FUNCTION_BLOCK FB_EventHandler IMPLEMENTS I_EventHandler
VAR_INPUT
END_VAR
VAR_OUTPUT
END_VAR
VAR
	// private instance var's
	iLog			: I_Logger;
	afbAlarm      	: ARRAY[0..Const.iMaxIdxAlam] OF FB_TcAlarm;
	fbCodeErrRef,
	fbAlarmRef      : REFERENCE TO FB_TcAlarm;
	fbMsg			: FB_TcMessage;
	fbEventLogger	: FB_TcEventLogger;
	ISb 			: I_StringBuilder;
	fbInternalSb	: FB_StringBuilder;
	iCntAlm			: INT;
	bInfoActive,
	bWarningActive,
	bErrorActive	: BOOL;
END_VAR

//ToDo: SetJsonAttribute (e.g.: error reaction)
//ToDo: F_GetEventText o.ä.
//ToDo: Listener?

// unit tests
Test();

METHOD PUBLIC ArgAddDint : I_EventHandler
VAR_INPUT
	value : DINT;
END_VAR
ArgAddDint := THIS^;
IF __ISVALIDREF(fbAlarmRef) THEN
	fbAlarmRef.ipArguments.AddDInt(value);
END_IF
END_METHOD

METHOD PUBLIC ArgAddEventRef : I_EventHandler
VAR_INPUT
	value : TcEventEntry;
END_VAR
ArgAddEventRef := THIS^;
IF __ISVALIDREF(fbAlarmRef) THEN
	fbAlarmRef.ipArguments.AddEventReferenceEx(value);
END_IF
END_METHOD

METHOD PUBLIC ArgAddLreal : I_EventHandler
VAR_INPUT
	value : LREAL;
END_VAR
ArgAddLreal := THIS^;
IF __ISVALIDREF(fbAlarmRef) THEN
	fbAlarmRef.ipArguments.AddLReal(value);
END_IF
END_METHOD

METHOD PUBLIC ArgAddString : I_EventHandler
VAR_IN_OUT CONSTANT
	value : STRING;
END_VAR
ArgAddString := THIS^;
IF __ISVALIDREF(fbAlarmRef) THEN
	fbAlarmRef.ipArguments.AddString(value);
END_IF
END_METHOD

METHOD PUBLIC ArgAddWString : I_EventHandler
VAR_IN_OUT CONSTANT
	value : WSTRING;
END_VAR
ArgAddWString := THIS^;
IF __ISVALIDREF(fbAlarmRef) THEN
	fbAlarmRef.ipArguments.AddWString(value);
END_IF
END_METHOD

METHOD PUBLIC ArgClear : I_EventHandler
ArgClear := THIS^;
IF __ISVALIDREF(fbAlarmRef) THEN
	fbAlarmRef.ipArguments.Clear();
END_IF
END_METHOD

METHOD PUBLIC ArgSbAppend : I_EventHandler
VAR_IN_OUT CONSTANT
	value : T_MaxString;
END_VAR
ArgSbAppend := THIS^;

IF ISb <> 0 THEN
	ISb.Append(value);
END_IF
END_METHOD

METHOD PUBLIC ArgSbAppendAny : I_EventHandler
VAR_INPUT
	value : ANY;
END_VAR
ArgSbAppendAny := THIS^;

IF ISb <> 0 THEN
	ISb.AppendAny(value);
END_IF
END_METHOD

METHOD PUBLIC ArgSbAppendAnyRaise : HRESULT
VAR_INPUT
	value : ANY;
END_VAR
ArgSbAppendAnyRaise := ArgSbAppendAny(value).ArgSetSbRaise();
END_METHOD

METHOD PUBLIC ArgSbAppendRaise : HRESULT
VAR_IN_OUT CONSTANT
	value : T_MaxString;
END_VAR
ArgSbAppendRaise := ArgSbAppendSet(value).Raise();
END_METHOD

METHOD PUBLIC ArgSbAppendS : I_EventHandler
VAR_INPUT
	value : T_MaxString := '';
END_VAR
ArgSbAppendS := ArgSbAppend(value);
END_METHOD

METHOD PUBLIC ArgSbAppendSet : I_EventHandler
VAR_IN_OUT CONSTANT
	value : T_MaxString;
END_VAR
ArgSbAppendSet := ArgSbAppend(value).ArgSetSb();
END_METHOD

METHOD PUBLIC ArgSbAppendWs : I_EventHandler
VAR_IN_OUT CONSTANT
	value : WSTRING;
END_VAR
ArgSbAppendWs := THIS^;

IF ISb <> 0 THEN
	ISb.AppendWs(value);
END_IF
END_METHOD

METHOD PUBLIC ArgSbAppendWsRaise : HRESULT
VAR_IN_OUT CONSTANT
	value : WSTRING;
END_VAR
ArgSbAppendWsRaise := ArgSbAppendWs(value).ArgSetSbRaise();
END_METHOD

METHOD PUBLIC ArgSbInit : I_EventHandler
VAR_IN_OUT CONSTANT
	value : T_MaxString;
END_VAR
Isb := fbInternalSb.Set(value);
ArgSbInit := THIS^;
END_METHOD

METHOD PUBLIC ArgSbInitExternal : I_EventHandler
VAR_INPUT
	sb	: I_StringBuilder;
END_VAR
ISb := sb;
ArgSbInitExternal := THIS^;
END_METHOD

METHOD PUBLIC ArgSbInitWs : I_EventHandler
VAR_IN_OUT CONSTANT
	value : WSTRING;
END_VAR
Isb := fbInternalSb.SetWs(value);
ArgSbInitWs := THIS^;
END_METHOD

METHOD PUBLIC ArgSetDint : I_EventHandler
VAR_INPUT
	value : DINT;
END_VAR
ArgSetDint := ArgClear().ArgAddDint(value);
END_METHOD

METHOD PUBLIC ArgSetEventRef : I_EventHandler
VAR_INPUT
	value : TcEventEntry;
END_VAR
ArgSetEventRef := ArgClear().ArgAddEventRef(value);
END_METHOD

METHOD PUBLIC ArgSetLreal : I_EventHandler
VAR_INPUT
	value : LREAL;
END_VAR
ArgSetLreal := ArgClear().ArgAddLreal(value);
END_METHOD

METHOD PUBLIC ArgSetSb : I_EventHandler
VAR_INPUT
	sb 		: I_StringBuilder := 0; // optional external string builder, set to 0 to use internal
END_VAR
VAR
	value	: STRING;
END_VAR
IF sb = 0 THEN
	sb := Isb;
END_IF

value := sb.ToString();
ArgSetSb := ArgClear().ArgAddString(value);
END_METHOD

METHOD PUBLIC ArgSetSbRaise : HRESULT
VAR_INPUT
	sb	: I_StringBuilder := 0; // optional external string builder, set to 0 to use internal
END_VAR
ArgSetSbRaise := ArgSetSb(sb).Raise();
END_METHOD

METHOD PUBLIC ArgSetString : I_EventHandler
VAR_IN_OUT CONSTANT
	value : STRING;
END_VAR
ArgSetString := ArgClear().ArgAddString(value);
END_METHOD

METHOD PUBLIC ArgSetWString : I_EventHandler
VAR_IN_OUT CONSTANT
	value : WSTRING;
END_VAR
ArgSetWString := ArgClear().ArgAddWString(value);
END_METHOD

METHOD PUBLIC CreateAlarm : I_EventHandler
VAR_INPUT
	stEventEntry      : TcEventEntry;
    bWithConfirmation : BOOL := FALSE;
    ipSourceInfo      : I_TcSourceInfo := NULL;
END_VAR
VAR
	hres 	: HRESULT;
	msg		: STRING;
END_VAR
CreateAlarm := THIS^;
IF (iCntAlm > Const.iMaxIdxAlam) THEN
	msg := CONCAT('Max. events exceeded, Const.iMaxIdxAlam: ', TO_STRING(Const.iMaxIdxAlam));
	fbCodeErrRef.ipArguments.Clear().AddString(msg);
	fbCodeErrRef.Raise(0);
	RETURN;
END_IF

hres := afbAlarm[iCntAlm].CreateEx(stEventEntry, bWithConfirmation, ipSourceInfo);

IF (hres = S_OK) THEN
	iCntAlm := iCntAlm + 1;
ELSE
	msg := CONCAT('Create alarm failed, HRESULT: ', TO_STRING(hres));
	fbCodeErrRef.ipArguments.Clear().AddString(msg);
	fbCodeErrRef.Raise(0);
END_IF
END_METHOD

{attribute 'monitoring' := 'call'}
PROPERTY ErrorActive : BOOL
GET
ErrorActive := bErrorActive;
END_GET
END_PROPERTY

{attribute 'monitoring' := 'call'}
PROPERTY InfoActive : BOOL
GET
InfoActive := bInfoActive;
END_GET
END_PROPERTY

METHOD Init : BOOL
iLog := SERVICES.ILog;

// init alarm event classes
CreateAlarm(TC_Events.InternalEventClass.InfoEvent);
CreateAlarm(TC_Events.InternalEventClass.WarningEvent, TRUE);
CreateAlarm(TC_Events.InternalEventClass.ErrorEvent, TRUE);
CreateAlarm(TC_Events.CodeEventClass.InfoEvent);
CreateAlarm(TC_Events.CodeEventClass.WarningEvent, TRUE);
CreateAlarm(TC_Events.CodeEventClass.ErrorEvent, TRUE);
CreateAlarm(TC_Events.SystemEventClass.InfoEvent);
CreateAlarm(TC_Events.SystemEventClass.WarningEvent, TRUE);
CreateAlarm(TC_Events.SystemEventClass.ErrorEvent, TRUE);
CreateAlarm(TC_Events.EtherCatEventClass.InfoEvent);
CreateAlarm(TC_Events.EtherCatEventClass.WarningEvent, TRUE);
CreateAlarm(TC_Events.EtherCatEventClass.ErrorEvent, TRUE);
CreateAlarm(TC_Events.EtherCatEventClass.DevicStateErrorEvent, TRUE);
CreateAlarm(TC_Events.EtherCatEventClass.LinkStateErrorEvent, TRUE);
CreateAlarm(TC_Events.HardwareEventClass.InfoEvent);
CreateAlarm(TC_Events.HardwareEventClass.WarningEvent, TRUE);
CreateAlarm(TC_Events.HardwareEventClass.ErrorEvent, TRUE);
CreateAlarm(TC_Events.TwinSafeEventClass.InfoEvent);
CreateAlarm(TC_Events.TwinSafeEventClass.WarningEvent, TRUE);
CreateAlarm(TC_Events.TwinSafeEventClass.ErrorEvent, TRUE);
CreateAlarm(TC_Events.TwinSafeEventClass.HwErrorEvent, TRUE);
CreateAlarm(TC_Events.SettingsEventClass.InfoEvent);
CreateAlarm(TC_Events.SettingsEventClass.WarningEvent, TRUE);
CreateAlarm(TC_Events.SettingsEventClass.ErrorEvent, TRUE);
CreateAlarm(TC_Events.RecipeEventClass.InfoEvent);
CreateAlarm(TC_Events.RecipeEventClass.WarningEvent, TRUE);
CreateAlarm(TC_Events.RecipeEventClass.ErrorEvent, TRUE);
CreateAlarm(TC_Events.PlantEventClass.InfoEvent);
CreateAlarm(TC_Events.PlantEventClass.WarningEvent, TRUE);
CreateAlarm(TC_Events.PlantEventClass.ErrorEvent, TRUE);

// register simple message not needed:
//CreateMessage(TC_Events.MessageEventClass.InfoEvent);

fbCodeErrRef REF= afbAlarm[0];
fbAlarmRef REF= afbAlarm[0];
END_METHOD

METHOD PUBLIC Raise : HRESULT
VAR_INPUT
	nTimeStamp : ULINT := 0;
END_VAR
IF NOT __ISVALIDREF(fbAlarmref) THEN 
	Raise := S_FALSE;
	RETURN;	
END_IF

bInfoActive := fbAlarmRef.eSeverity >= TcEventSeverity.Info;
bWarningActive := fbAlarmRef.eSeverity >= TcEventSeverity.Warning;
bErrorActive := fbAlarmRef.eSeverity >= TcEventSeverity.Error;
Raise := fbAlarmref.Raise(nTimeStamp);
END_METHOD

METHOD PUBLIC Reset : BOOL
VAR_INPUT
END_VAR
fbEventLogger.ConfirmAllAlarms();
fbEventLogger.ClearAllAlarms();
fbEventLogger.ClearLoggedEvents(0);

bInfoActive :=
bWarningActive :=
bErrorActive := FALSE;
END_METHOD

METHOD PUBLIC Select : I_EventHandler
VAR_INPUT
	stEventEntry : TcEventEntry;
END_VAR
VAR
	hres : HRESULT;
END_VAR
Select := THIS^;
fbAlarmRef REF= afbAlarm[0];
hres := fbEventLogger.GetAlarmEx(stEventEntry, 0, fbAlarmRef);
IF hres <> S_OK OR NOT __ISVALIDREF(fbAlarmRef) THEN
	fbAlarmRef REF= afbAlarm[0];
END_IF
END_METHOD

METHOD PUBLIC Send : BOOL
VAR_INPUT
	stEventEntry      : TcEventEntry;
    ipSourceInfo      : I_TcSourceInfo := NULL;
    nTimeStamp        : ULINT := 0;
    ipArguments       : I_TcArguments := NULL;
END_VAR
Send := fbEventLogger.SendMessageEx(stEventEntry, ipSourceInfo, nTimeStamp, ipArguments) = S_OK;
END_METHOD

METHOD PUBLIC SendJson : BOOL
VAR_INPUT
	stEventEntry      : TcEventEntry;
    ipSourceInfo      : I_TcSourceInfo := NULL;
    nTimeStamp        : ULINT := 0;
    ipArguments       : I_TcArguments := NULL;
END_VAR
VAR_IN_OUT CONSTANT
    sJsonAttribute    : STRING;
END_VAR
SendJson := fbEventLogger.SendMessageEx2(stEventEntry, ipSourceInfo, nTimeStamp, ipArguments, sJsonAttribute) = S_OK;
END_METHOD

METHOD PUBLIC SendString : BOOL
VAR_IN_OUT CONSTANT
	msg : STRING;	
END_VAR
VAR_INST
	args : FB_TcArguments;
END_VAR
SendString := Send(TC_EVENTS.MessageEventClass.InfoEvent, NULL, 0, 
													args.Clear().AddString(msg));
END_METHOD

METHOD PUBLIC SendStringJson : BOOL
VAR_IN_OUT CONSTANT
	msg				: STRING;
	sJsonAttribute	: STRING;
END_VAR
VAR_INST
	args 			: FB_TcArguments;
END_VAR
SendStringJson := SendJson(TC_EVENTS.MessageEventClass.InfoEvent, NULL, 0, 
													args.Clear().AddString(msg), 
													sJsonAttribute);
END_METHOD

METHOD PRIVATE Test : BOOL
VAR_INST
	// event alarm test
	iTestCase		: INT;
	bAlarmTest, 
	bMsgTest,
	bClearAlarmTest : BOOL;
	HRES			: HRESULT;
END_VAR
// alarm tests
IF bAlarmTest THEN
	bAlarmTest := FALSE;
	IF iTestCase = 0 THEN
		HRES := fbEventLogger.GetAlarmEx(TC_Events.CodeEventClass.ErrorEvent, 0, fbAlarmRef);
		IF (HRES <> 0 OR  NOT __ISVALIDREF(fbAlarmRef)) THEN RETURN; END_IF
		iTestCase := 10;
		fbAlarmRef.ipArguments.Clear().AddString('check bounds');
		fbAlarmRef.Raise(0);
		
	ELSIF iTestCase = 1 THEN
		Select(TC_Events.CodeEventClass.ErrorEvent)
			  .ArgSetString('check bounds')
			  .Raise();
		RETURN;
	ELSIF iTestCase = 2 THEN
		Select(TC_Events.HardwareEventClass.ErrorEvent)
			  .ArgSetString('div 0')
			  .Raise();
	ELSIF iTestCase = 3 THEN		
		Select(TC_Events.HardwareEventClass.WarningEvent)
			  .ArgSetString('check pointer')
			  .Raise();
	ELSIF iTestCase = 4 THEN
		// adding localizable argument sample 
		Select(TC_Events.SettingsEventClass.InfoEvent)
			  .ArgSetEventRef(TC_Events.TranslationListEventClass.TranslationListEventClass_NameEvent)
			  .ArgAddString('sdc')
			  .Raise();
	END_IF
	
	//fbAlarm.eConfirmationState = TcEventConfirmationState.WaitForConfirmation
	//fbAlarm.bActive
END_IF

// simple message tests
IF bMsgTest THEN
	bMsgTest := FALSE;
	IF iTestCase = 0 THEN
		SendString('Rezept wurde geladen!');
	ELSIF iTestCase = 2 THEN
		SendString('Rezept wurde gespeichert!');
	ELSIF iTestCase = 3 THEN
		SendString('Rezept wurde kopiert!');
	ELSE
		Send(TC_Events.MessageEventClass.InfoEvent, Null, 0, fbMsg.ipArguments);
	END_IF
	
	//fbMsg.Send();
END_IF

// reset/clear alarms
IF bClearAlarmTest THEN
	bClearAlarmTest := FALSE;
	Reset();
END_IF
END_METHOD

{attribute 'monitoring' := 'call'}
PROPERTY WarningActive : BOOL
GET
WarningActive := bWarningActive;
END_GET
END_PROPERTY

END_FUNCTION_BLOCK

(* stored: Version 1.1.0.1
   POU FB_EventHandler: Id {15ddc12e-d496-402a-851f-a36d0274e1a7}, SpecialFunc None
   Folder Fluent: Id {d2bbe7f3-5e4b-4cc3-aa32-c720a5287f9b}
   Folder StringBuilder: Id {fcbc0fab-a6db-4129-b0c7-3a0281c2e83b}
   Folder Properties: Id {63e5b720-7618-4c1a-b230-482d965e0c2d}
   Folder SimpleMsg: Id {ae694419-03a6-450d-b02e-b681c0ee8f90}
   Method ArgAddDint: Id {a0f05de7-44e2-4def-b35f-8d4f1a855e11}
   Method ArgAddEventRef: Id {6d53bd2d-6ff4-4620-a3f0-cd16b37035a0}
   Method ArgAddLreal: Id {f58f88ba-eecf-4ee6-93c3-f50790edaf05}
   Method ArgAddString: Id {b7defce1-c44c-4877-b18a-8de91a9a0687}
   Method ArgAddWString: Id {df6e7669-76f4-40f3-9750-93822785ae03}
   Method ArgClear: Id {711b7cb5-ea45-4174-91b9-167f83a91498}
   Method ArgSbAppend: Id {d2d4a8c9-c966-4d76-a27f-1661401580a3}
   Method ArgSbAppendAny: Id {7bc07fa3-be49-444a-b032-24ce77801483}
   Method ArgSbAppendAnyRaise: Id {a814fe43-1556-4b26-bf00-8661f391cd0c}
   Method ArgSbAppendRaise: Id {5a237caa-ae8e-46c8-a87e-08d50843e498}
   Method ArgSbAppendS: Id {3c65e138-dbf6-4ed5-aaee-5912040b50c7}
   Method ArgSbAppendSet: Id {b46737c0-41fd-4660-b440-0b0fa7c2152b}
   Method ArgSbAppendWs: Id {f3f16ae3-4024-4f3e-a07d-a8e4fc39c782}
   Method ArgSbAppendWsRaise: Id {e2782b5b-50a6-430e-b3db-8126b33ea375}
   Method ArgSbInit: Id {b1ec0e9a-05cb-493e-96e3-206a1518a5d4}
   Method ArgSbInitExternal: Id {355f971e-a413-454f-b883-bdb8992cbb7c}
   Method ArgSbInitWs: Id {f2bae4ed-ebcb-40eb-8c0b-35ec9dea60ce}
   Method ArgSetDint: Id {5afe283e-bc59-4fa2-b13a-bbc0c036bb15}
   Method ArgSetEventRef: Id {bc16718f-95fc-4020-be08-dda3136e53e7}
   Method ArgSetLreal: Id {f33f133a-277d-4ddf-80b9-d8e30b421a13}
   Method ArgSetSb: Id {e2cf4d4e-36ca-4e85-a6bf-fd4680840585}
   Method ArgSetSbRaise: Id {fa5c1d0e-634f-476e-984e-f0c8181a0e57}
   Method ArgSetString: Id {a70b022b-ab77-40f4-b874-0d6d5e6d1a48}
   Method ArgSetWString: Id {7f3a8654-472d-488f-98bb-f06bc8c61fcc}
   Method CreateAlarm: Id {1f60ac4f-2e26-4b3b-8d04-66a211566c2d}
   Property ErrorActive: Id {0e6431d2-f8db-4726-8b67-e4d53b5c74be}
   Get Get: Id {f0fa74ee-b95e-4d22-975a-e1578c84fd38}
   Property InfoActive: Id {00622ccf-c6d3-491f-aaaa-96ee484f4af0}
   Get Get: Id {b33334a8-5d23-4c9e-92a7-5e1ba2424e3c}
   Method Init: Id {fb7a6f7b-d623-47ab-8142-e647ea1a6022}
   Method Raise: Id {e70de61e-a502-44e9-a48e-2cdfab490faf}
   Method Reset: Id {d27a7122-a7a6-4cac-bd3d-60c72f3b7d27}
   Method Select: Id {acc4527b-aa49-4a3f-8e5a-cc2218a63cc8}
   Method Send: Id {fce0bd20-fde8-463f-b238-4262ebb02044}
   Method SendJson: Id {4f727c5f-68e6-4b53-93ea-43be75604602}
   Method SendString: Id {7740b874-26f7-4c93-aad8-6040f7f3132e}
   Method SendStringJson: Id {e92fa693-1d37-401f-85b1-1d4c3a1d5fc4}
   Method Test: Id {6dd5f8ba-68eb-4a0b-b379-52cf1523025c}
   Property WarningActive: Id {9509dd0d-e8b6-4af2-8ece-e73686062c40}
   Get Get: Id {857e3c4c-42cb-46f6-9c65-a463c6ce1bed} *)
